# EPICS autosave request: valon5009App/Db/valon5009_settings.req
# This file specifies which PVs of the corresponding database should be saved.

# Output Power
$(P)$(R)Src1Pwr-SP
$(P)$(R)Src2Pwr-SP

# Output Frequency
$(P)$(R)Src1Freq-SP
$(P)$(R)Src2Freq-SP

# Output Frequency Offset
$(P)$(R)Src1FreqOffset-SP
$(P)$(R)Src2FreqOffset-SP

# Attenuator
$(P)$(R)AttenuatorStep-Cte
$(P)$(R)Src1Attenuator-SP
$(P)$(R)Src2Attenuator-SP

# Power Level
$(P)$(R)Src1PwrLvl-Sel
$(P)$(R)Src2PwrLvl-Sel

# Enable Output Buffer Amplifier
$(P)$(R)BuffAmpGain-Cte
$(P)$(R)Src1EnblBuffAmp-Sel
$(P)$(R)Src2EnblBuffAmp-Sel

# Power Down Source
$(P)$(R)Src1PwrOn-Sel
$(P)$(R)Src2PwrOn-Sel

# Reference settings
$(P)$(R)RefFreq-SP
$(P)$(R)RefTrim-SP
$(P)$(R)RefSrcType-Sel

# Reference PFD
$(P)$(R)Src1PFD-SP
$(P)$(R)Src2PFD-SP

# Reference Doubler
$(P)$(R)Src1RefDoubler-Sel
$(P)$(R)Src2RefDoubler-Sel

# Reference Divider
$(P)$(R)Src1RefDivider-Sel
$(P)$(R)Src2RefDivider-Sel
